// Mitsubishi GX Works2 project: 세탁기2   PLC: Q03UDV

PROGRAM MAIN
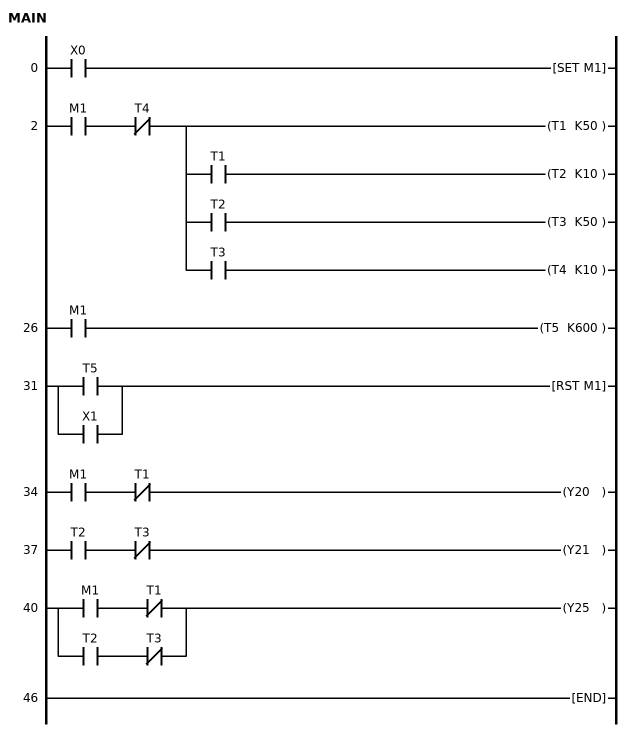
0     LD      X0
      SET     M1
2     LD      M1
      ANI     T4
      OUT     T1 K50
      MPS
      AND     T1
      OUT     T2 K10
      MRD
      AND     T2
      OUT     T3 K50
      MPP
      AND     T3
      OUT     T4 K10
26    LD      M1
      OUT     T5 K600
31    LD      T5
      OR      X1
      RST     M1
34    LD      M1
      ANI     T1
      OUT     Y20
37    LD      T2
      ANI     T3
      OUT     Y21
40    LD      M1
      ANI     T1
      LD      T2
      ANI     T3
      ORB
      OUT     Y25
46    END
END_PROGRAM
